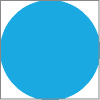
VISUALIZATION ButtonTemplate  // 100x100
VAR_IN_OUT
	bActive : BOOL;	
END_VAR
    Ellipse (0,0 100x100), colour toggle: bActive
    Ellipse (5,5 90x90)
END_VISUALIZATION

(* stored: Version 1.1.0.1, ProductVersion 3.1.4024.11
   Visu ButtonTemplate: Id {217189a3-2472-4d1c-bb5c-e8ea08153e46} *)
